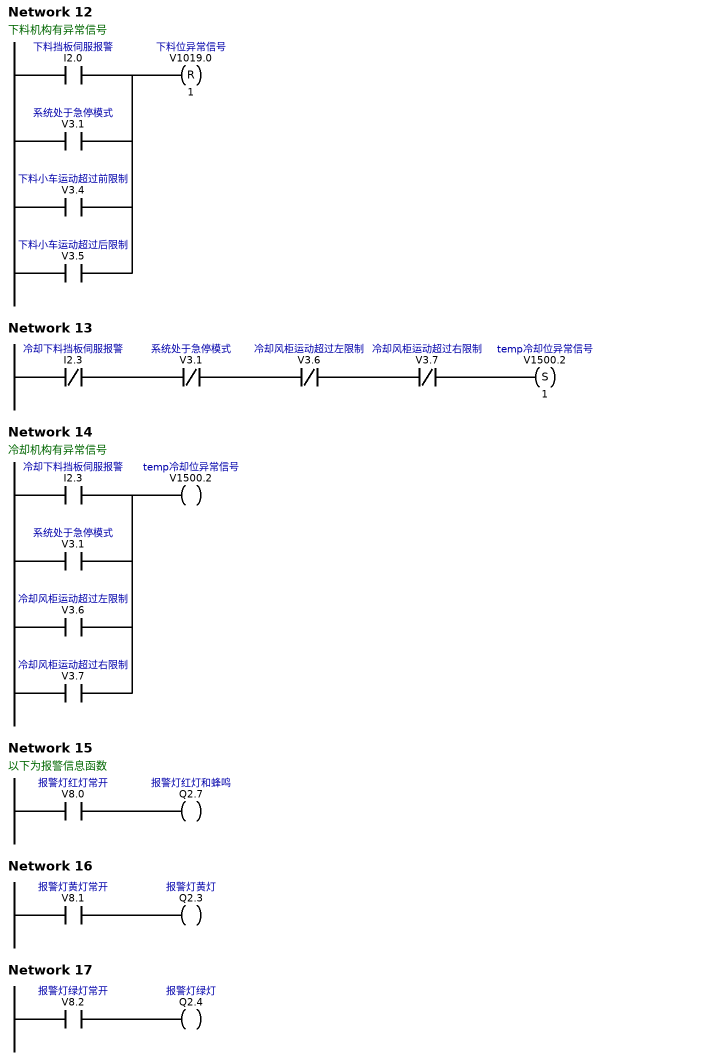
[picture p48: SBR21 networks 12-17]
Network 12
// 下料机构有异常信号
LD     下料挡板伺服报警:I2.0
O      系统处于急停模式:V3.1
O      下料小车运动超过前限制:V3.4
O      下料小车运动超过后限制:V3.5
R      下料位异常信号:V1019.0, 1
Network 13
LDN    冷却下料挡板伺服报警:I2.3
AN     系统处于急停模式:V3.1
AN     冷却风柜运动超过左限制:V3.6
AN     冷却风柜运动超过右限制:V3.7
S      temp冷却位异常信号:V1500.2, 1
Network 14
// 冷却机构有异常信号
LD     冷却下料挡板伺服报警:I2.3
O      系统处于急停模式:V3.1
O      冷却风柜运动超过左限制:V3.6
O      冷却风柜运动超过右限制:V3.7
=      temp冷却位异常信号:V1500.2
Network 15
// 以下为报警信息函数
LD     报警灯红灯常开:V8.0
=      报警灯红灯和蜂鸣:Q2.7
Network 16
LD     报警灯黄灯常开:V8.1
=      报警灯黄灯:Q2.3
Network 17
LD     报警灯绿灯常开:V8.2
=      报警灯绿灯:Q2.4
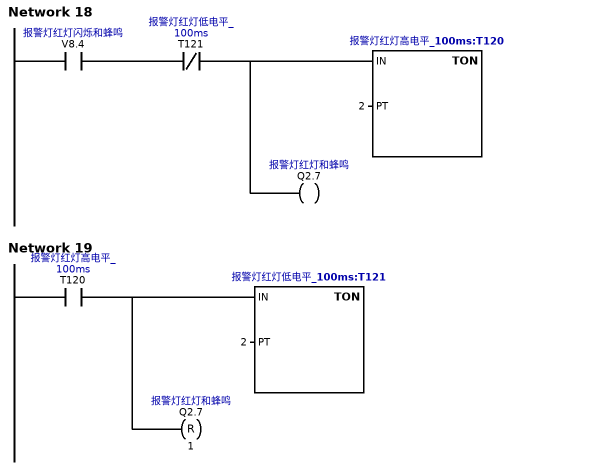
Network 18
LD     报警灯红灯闪烁和蜂鸣:V8.4
AN     报警灯红灯低电平_100ms:T121
TON    报警灯红灯高电平_100ms:T120, 2
=      报警灯红灯和蜂鸣:Q2.7
Network 19
LD     报警灯红灯高电平_100ms:T120
TON    报警灯红灯低电平_100ms:T121, 2
R      报警灯红灯和蜂鸣:Q2.7, 1
END_SUBROUTINE_BLOCK
